FUNCTION_BLOCK RIGHT (* IEC 61131-3,Table 29#3 *)
  (* Standard: 61131-3 *)
  (* Version 0.0, 2004-12-15, JHC, Rockwell Automation, Converted from SRC format. *)
  (* Compiler header: package fb.rt.plc.strings; *)
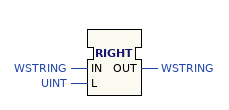
  VAR_INPUT
    IN : WSTRING;
    L : UINT;
  END_VAR
  VAR_OUTPUT
    OUT : WSTRING;
  END_VAR
END_FUNCTION_BLOCK
